FUNCTION_BLOCK ForeignCylinderControl (* Basic Function Block Type *)
  (* Standard: 61499-2 *)
  (* Version 0.0, 12/9/2021, e_net, nxtControl GmbH, Template *)
  PACKAGE Main;
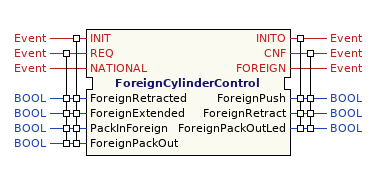
  EVENT_INPUT
    INIT WITH ForeignRetracted, ForeignExtended, PackInForeign, ForeignPackOut; (* Initialization Request *)
    REQ WITH ForeignRetracted, ForeignExtended, PackInForeign, ForeignPackOut; (* Normal Execution Request *)
    NATIONAL;
  END_EVENT
  EVENT_OUTPUT
    INITO WITH ForeignPush, ForeignRetract, ForeignPackOutLed; (* Initialization Confirm *)
    CNF WITH ForeignPush, ForeignRetract, ForeignPackOutLed; (* Execution Confirmation *)
    FOREIGN;
  END_EVENT
  VAR_INPUT
    ForeignRetracted : BOOL;
    ForeignExtended : BOOL;
    PackInForeign : BOOL;
    ForeignPackOut : BOOL;
  END_VAR
  VAR_OUTPUT
    ForeignPush : BOOL;
    ForeignRetract : BOOL;
    ForeignPackOutLed : BOOL;
  END_VAR
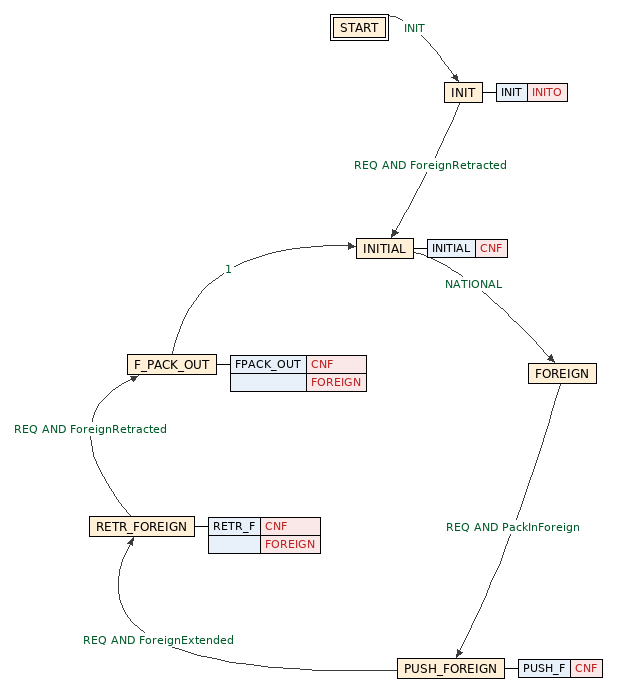
  EC_STATES
    START; (* Initial State *)
    INIT : INIT -> INITO; (* Initialization *)
    INITIAL : INITIAL -> CNF;
    PUSH_FOREIGN : PUSH_F -> CNF;
    RETR_FOREIGN : RETR_F -> CNF, -> FOREIGN;
    F_PACK_OUT : FPACK_OUT -> CNF, -> FOREIGN;
    FOREIGN;
  END_STATES
  EC_TRANSITIONS
    START TO INIT := INIT;
    INIT TO INITIAL := REQ AND ForeignRetracted;
    FOREIGN TO PUSH_FOREIGN := REQ AND PackInForeign;
    PUSH_FOREIGN TO RETR_FOREIGN := REQ AND ForeignExtended;
    RETR_FOREIGN TO F_PACK_OUT := REQ AND ForeignRetracted;
    F_PACK_OUT TO INITIAL := 1;
    INITIAL TO FOREIGN := NATIONAL;
  END_TRANSITIONS
  ALGORITHM INIT IN ST: (* Initialization algorithm *)
ForeignPush:= FALSE;
ForeignRetract:= TRUE;
  END_ALGORITHM
  ALGORITHM INITIAL IN ST:
ForeignRetract:=FALSE;
  END_ALGORITHM
  ALGORITHM PUSH_F IN ST:
ForeignPush:=TRUE;
ForeignPackOutLed:=TRUE;
  END_ALGORITHM
  ALGORITHM RETR_F IN ST:
ForeignPush:=FALSE;
ForeignRetract:=TRUE;
  END_ALGORITHM
  ALGORITHM FPACK_OUT IN ST:
ForeignPackOutLed:=FALSE;
  END_ALGORITHM
END_FUNCTION_BLOCK
